FUNCTION ASCF_CL_104_IF5 : Word
VAR_OUTPUT
	Out						: ASCF_UnionType;				//Result of the computation (Type: VDWord)
END_VAR

VAR_IN_OUT
	Arguments				: ARRAY[0..3] OF ASCF_UnionType;	//Arguments for the function (Argument[0]: VDWord, Argument[1]: VDWord, Argument[2]: VDWord, Argument[3]: VDWord)
	Memory					: ASCF_CL_ArgumentType;				//Memory to store data
END_VAR

VAR
	State1					: DWORD;
	State2					: DWORD;
	Command					: DWORD;
	PrevCommand				: DWORD;
	tempQCs					: ARRAY[0..3] OF BYTE;
	constDefaultUnionType	: ASCF_UnionType;				//Union type that holds only one of its possible data types at a time. The type can be selected via the "Typeselector". Independent of the selected type, every value has a quality code "VQC".
	constUnionTypes			: ASCF_EnumUnionTypes;			//Enumeration type of the valid values for the "Typeselector" of a "GVR_unionType"-UDT.
	constQualityCodes		: ASCF_QualityCodes;				//This enum encodes the defines quality codes for the MTP standard. The values are shown in HEX. The lowest value (1) has the highest priority.    | QC Name              | Value | Priority ||----------------------|:-----:|:--------:|| Failure              | 16#00 |    1     || Function Check       | 16#60 |    2     || Ma: INTenance Request  | 16#A4 |    3     || Out of Specification | 16#68 |    4     || OK                   | 16#80 |    5     || Out of Service       | 16#1C |    6     || No Status            | 16#FF |    7     |
	constSourceTypes		: ASCF_CL_EnumSourceTypes;			//Enumeration of source types of the Adaptive Logic.
	constErrors				: ASCF_CL_EnumErrors;				//Enumeration type of the error codes of the Adaptive Logic.
END_VAR



//#################################################################################################
{region "INITIALIZE VARIABLES"}
    Out := constDefaultUnionType;
{endregion}

//#################################################################################################
{region "CHECK ARG0"}
    // Arg0.Source can't be "Constant" because it's used to store the
    // result of this cycle to detect a possible edge in the next cycle
    IF Memory.Source = constSourceTypes.Constante THEN
        ASCF_CL_104_IF5 := constErrors.InvalidSourceSelected;
    END_IF;
{endregion}

//#################################################################################################
{region "PROCESS ARGUMENTS"}
    //-------------------------------------------------------------------------------------
    // State 1
    IF Arguments[0].Typeselector <> constUnionTypes.VDWord THEN
        ASCF_CL_104_IF5 := constErrors.InvalidType;
        RETURN;
    END_IF;
    
    //-------------------------------------------------------------------------------------
    // State 2
    IF Arguments[1].Typeselector <> constUnionTypes.VDWord THEN
        ASCF_CL_104_IF5 := constErrors.InvalidType;
        RETURN;
    END_IF;
    
    //-------------------------------------------------------------------------------------
    // Command
    IF Arguments[2].Typeselector <> constUnionTypes.VDWord THEN
        ASCF_CL_104_IF5 := constErrors.InvalidType;
        RETURN;
    END_IF;
    
    //-------------------------------------------------------------------------------------
    // Previous Command
    IF Arguments[3].Typeselector <> constUnionTypes.VDWord THEN
        ASCF_CL_104_IF5 := constErrors.InvalidType;
        RETURN;
    END_IF;
    
    State1 := Arguments[0].VDWord;
    State2 := Arguments[1].VDWord;
    Command := Arguments[2].VDWord;
    PrevCommand := Arguments[3].VDWord;
    tempQCs[0] := Arguments[0].VQC;
    tempQCs[1] := Arguments[1].VQC;
    tempQCs[2] := Arguments[2].VQC;
    tempQCs[3] := Arguments[3].VQC;
{endregion}

//#################################################################################################
{region "OUTPUT"}
    Out.VQC := ASCF_CalcWQC(QC1 := ASCF_CalcWQC(QC1 := tempQCs[0], QC2 := tempQCs[1]), QC2 := ASCF_CalcWQC(QC1 := tempQCs[2], QC2 := tempQCs[3]));
    Out.Typeselector := constUnionTypes.VDWord;
    
    IF State1 <> State2 AND Memory.Const.VBool THEN
        Out.VDWord := Command;
        
    ELSE
        Out.VDWord := PrevCommand;
        
    END_IF;
    
    Memory.Const.VBool := State1 = State2;
    
    ASCF_CL_104_IF5 := constErrors.None;
{endregion}

END_FUNCTION

(* stored: Version 1.1.0.1, ProductVersion 3.1.4026.4
   POU ASCF_CL_104_IF5: Id {b85544c2-b25a-47fe-960b-4d173f987557}, SpecialFunc None *)
